FUNCTION proj4_TupleStruct_1: REAL
{ S7_Optimized_Access := 'false' }
    VAR_INPUT
        tuple: TupleStruct_1;
    END_VAR

BEGIN
    proj4_TupleStruct_1 := tuple.field4;
END_FUNCTION
